// TIA Portal V21 export
TYPE "Std_DispositivoProfinet"
   STRUCT
      Allarmi : Struct
         "A" : Array[0.."K_NumAllarmiPerDispositivoProfinet"] of "Std_PrmAllarmeStd";
         WordHMI { S7_SetPoint := 'True'} : Word;
      END_STRUCT;
   END_STRUCT;
END_TYPE
